// TIA Portal V17 export
// export: Created 2022-07-20T06:59:49.9012984Z, ExportSetting WithDefaults, DisplayName Totally Integrated Automation Portal, DisplayVersion V17, DisplayName TIA Portal Openness, DisplayVersion V17, DisplayName TIA Portal Version Control Interface, DisplayVersion V17, DisplayName SINAMICS Startdrive Advanced, DisplayVersion V17, DisplayName SINAMICS Startdrive G130, G150, S120, S150, SINAMICS MV, S210, DisplayVersion V17, DisplayName SINAMICS Startdrive G110M, G120, G120C, G120D, G120P, G115D, DisplayVersion V17, DisplayName STEP 7 Professional, DisplayVersion V17, DisplayName STEP 7 Safety, DisplayVersion V17, DisplayName WinCC Advanced, DisplayVersion V17
FUNCTION "FC10024_ArrayAverage" : Void   // FC10024, LAD
{ S7_Optimized_Access := 'TRUE' }
VERSION : 0.1
// stored: AutoNumber false, IsIECCheckEnabled false, SetENOAutomatically false, UDAEnableTagReadback false
   VAR_INPUT
      "Array" : Array[*] of LReal;
      NumberOfValues : Int;
   END_VAR
   VAR_OUTPUT
      Average : LReal;
   END_VAR
   VAR_TEMP
      i : Int;
      Sum : LReal;
   END_VAR
BEGIN

REGION Network 1 (SCL): Calculation Of The Average
   FOR #i := 0 TO #NumberOfValues - 1 DO
       #Sum += #Array[#i];
   END_FOR;
   #Average := #Sum / INT_TO_LREAL(#NumberOfValues);
END_REGION
END_FUNCTION
